KUKA KRL program: Kuka_Relative_Mo2.src

&ACCESS RVP
&REL 1
&PARAM TEMPLATE = C:\KRC\Roboter\Template\vorgabe
&PARAM EDITMASK = *
DEF Kuka_Relative_Mo2 ( )
; TOOL_DATA[1] = {FRAME: X 0.000,Y 0.000,Z 10.000,A 0.000,B 0.000,C 0.000}
$TOOL = {FRAME: X 0.000,Y 0.000,Z 10.000,A 0.000,B 0.000,C 0.000}
; $TOOL = TOOL_DATA[1]
; --------------------------
PTP {A1 -91.15290,A2 -57.66310,A3 113.87200,A4 27.68180,A5 -61.31820,A6 -12.21360}
; ---- Setting reference (Base) ----
$BASE = {FRAME: X 0.000,Y 0.000,Z 0.000,A 0.000,B 0.000,C 0.000}
; --------------------------
; ---- Setting tool (TCP) ----
; TOOL_DATA[1] = {FRAME: X 0.000,Y 0.000,Z 10.000,A 0.000,B 0.000,C 0.000}
$TOOL = {FRAME: X 0.000,Y 0.000,Z 10.000,A 0.000,B 0.000,C 0.000}
; $TOOL = TOOL_DATA[1]
; --------------------------
PTP {A1 -96.29580,A2 -57.85820,A3 114.83400,A4 -12.72140,A5 -60.67670,A6 8.34871}
; ---- Setting reference (Base) ----
$BASE = {FRAME: X 0.000,Y 0.000,Z 0.000,A 0.000,B 0.000,C 0.000}
; --------------------------
; ---- Setting tool (TCP) ----
; TOOL_DATA[1] = {FRAME: X 0.000,Y 0.000,Z 10.000,A 0.000,B 0.000,C 0.000}
$TOOL = {FRAME: X 0.000,Y 0.000,Z 10.000,A 0.000,B 0.000,C 0.000}
; $TOOL = TOOL_DATA[1]
; --------------------------
PTP {A1 -96.29580,A2 -57.85820,A3 114.83400,A4 -12.72140,A5 -60.67670,A6 -21.65130}
; ---- Setting reference (Base) ----
$BASE = {FRAME: X 0.000,Y 0.000,Z 0.000,A 0.000,B 0.000,C 0.000}
; --------------------------
; ---- Setting tool (TCP) ----
; TOOL_DATA[1] = {FRAME: X 0.000,Y 0.000,Z 10.000,A 0.000,B 0.000,C 0.000}
$TOOL = {FRAME: X 0.000,Y 0.000,Z 10.000,A 0.000,B 0.000,C 0.000}
; $TOOL = TOOL_DATA[1]
; --------------------------
PTP {A1 -96.29580,A2 -57.85820,A3 114.83400,A4 -12.72140,A5 -60.67670,A6 38.34870}
; ---- Setting reference (Base) ----
$BASE = {FRAME: X 0.000,Y 0.000,Z 0.000,A 0.000,B 0.000,C 0.000}
; --------------------------
; ---- Setting tool (TCP) ----
; TOOL_DATA[1] = {FRAME: X 0.000,Y 0.000,Z 10.000,A 0.000,B 0.000,C 0.000}
$TOOL = {FRAME: X 0.000,Y 0.000,Z 10.000,A 0.000,B 0.000,C 0.000}
; $TOOL = TOOL_DATA[1]
; --------------------------
PTP {A1 -96.29580,A2 -57.85820,A3 114.83400,A4 -12.72140,A5 -60.67670,A6 8.34871}
; ---- Setting reference (Base) ----
$BASE = {FRAME: X 0.000,Y 0.000,Z 0.000,A 0.000,B 0.000,C 0.000}
; --------------------------
; ---- Setting tool (TCP) ----
; TOOL_DATA[1] = {FRAME: X 0.000,Y 0.000,Z 10.000,A 0.000,B 0.000,C 0.000}
$TOOL = {FRAME: X 0.000,Y 0.000,Z 10.000,A 0.000,B 0.000,C 0.000}
; $TOOL = TOOL_DATA[1]
; --------------------------
PTP {A1 -85.43380,A2 -57.35410,A3 116.48600,A4 -0.25181,A5 -62.16390,A6 1.57543}
; ---- Setting reference (Base) ----
$BASE = {FRAME: X 0.000,Y 0.000,Z 0.000,A 0.000,B 0.000,C 0.000}
; --------------------------
; ---- Setting tool (TCP) ----
; TOOL_DATA[1] = {FRAME: X 0.000,Y 0.000,Z 10.000,A 0.000,B 0.000,C 0.000}
$TOOL = {FRAME: X 0.000,Y 0.000,Z 10.000,A 0.000,B 0.000,C 0.000}
; $TOOL = TOOL_DATA[1]
; --------------------------
PTP {A1 -90.40980,A2 -56.06330,A3 113.85800,A4 -38.62590,A5 -67.35010,A6 19.20140}
; ---- Setting reference (Base) ----
$BASE = {FRAME: X 0.000,Y 0.000,Z 0.000,A 0.000,B 0.000,C 0.000}
; --------------------------
; ---- Setting tool (TCP) ----
; TOOL_DATA[1] = {FRAME: X 0.000,Y 0.000,Z 10.000,A 0.000,B 0.000,C 0.000}
$TOOL = {FRAME: X 0.000,Y 0.000,Z 10.000,A 0.000,B 0.000,C 0.000}
; $TOOL = TOOL_DATA[1]
; --------------------------
PTP {A1 -80.44290,A2 -56.45170,A3 113.95500,A4 38.75120,A5 -65.60370,A6 -16.89390}
; ---- Setting reference (Base) ----
$BASE = {FRAME: X 0.000,Y 0.000,Z 0.000,A 0.000,B 0.000,C 0.000}
; --------------------------
; ---- Setting tool (TCP) ----
; TOOL_DATA[1] = {FRAME: X 0.000,Y 0.000,Z 10.000,A 0.000,B 0.000,C 0.000}
$TOOL = {FRAME: X 0.000,Y 0.000,Z 10.000,A 0.000,B 0.000,C 0.000}
; $TOOL = TOOL_DATA[1]
; --------------------------
PTP {A1 -85.43380,A2 -57.35410,A3 116.48600,A4 -0.25181,A5 -62.16390,A6 1.57543}
; ---- Setting reference (Base) ----
$BASE = {FRAME: X 0.000,Y 0.000,Z 0.000,A 0.000,B 0.000,C 0.000}
; --------------------------
; ---- Setting tool (TCP) ----
; TOOL_DATA[1] = {FRAME: X 0.000,Y 0.000,Z 10.000,A 0.000,B 0.000,C 0.000}
$TOOL = {FRAME: X 0.000,Y 0.000,Z 10.000,A 0.000,B 0.000,C 0.000}
; $TOOL = TOOL_DATA[1]
; --------------------------
PTP {A1 -85.43380,A2 -57.35410,A3 116.48600,A4 -0.25181,A5 -62.16390,A6 -28.42460}
; ---- Setting reference (Base) ----
$BASE = {FRAME: X 0.000,Y 0.000,Z 0.000,A 0.000,B 0.000,C 0.000}
; --------------------------
; ---- Setting tool (TCP) ----
; TOOL_DATA[1] = {FRAME: X 0.000,Y 0.000,Z 10.000,A 0.000,B 0.000,C 0.000}
$TOOL = {FRAME: X 0.000,Y 0.000,Z 10.000,A 0.000,B 0.000,C 0.000}
; $TOOL = TOOL_DATA[1]
; --------------------------
PTP {A1 -85.43380,A2 -57.35410,A3 116.48600,A4 -0.25181,A5 -62.16390,A6 31.57540}
; ---- Setting reference (Base) ----
$BASE = {FRAME: X 0.000,Y 0.000,Z 0.000,A 0.000,B 0.000,C 0.000}
; --------------------------
; ---- Setting tool (TCP) ----
; TOOL_DATA[1] = {FRAME: X 0.000,Y 0.000,Z 10.000,A 0.000,B 0.000,C 0.000}
$TOOL = {FRAME: X 0.000,Y 0.000,Z 10.000,A 0.000,B 0.000,C 0.000}
; $TOOL = TOOL_DATA[1]
; --------------------------
PTP {A1 -85.43380,A2 -57.35410,A3 116.48600,A4 -0.25181,A5 -62.16390,A6 1.57543}
; ---- Setting reference (Base) ----
$BASE = {FRAME: X 0.000,Y 0.000,Z 0.000,A 0.000,B 0.000,C 0.000}
; --------------------------
; ---- Setting tool (TCP) ----
; TOOL_DATA[1] = {FRAME: X 0.000,Y 0.000,Z 10.000,A 0.000,B 0.000,C 0.000}
$TOOL = {FRAME: X 0.000,Y 0.000,Z 10.000,A 0.000,B 0.000,C 0.000}
; $TOOL = TOOL_DATA[1]
; --------------------------
PTP {A1 -86.65140,A2 -57.29670,A3 116.45300,A4 -1.62638,A5 -62.19900,A6 2.28097}
; ---- Setting reference (Base) ----
$BASE = {FRAME: X 0.000,Y 0.000,Z 0.000,A 0.000,B 0.000,C 0.000}
; --------------------------
; ---- Setting tool (TCP) ----
; TOOL_DATA[1] = {FRAME: X 0.000,Y 0.000,Z 10.000,A 0.000,B 0.000,C 0.000}
$TOOL = {FRAME: X 0.000,Y 0.000,Z 10.000,A 0.000,B 0.000,C 0.000}
; $TOOL = TOOL_DATA[1]
; --------------------------
PTP {A1 -91.58690,A2 -55.92760,A3 113.65300,A4 -39.84090,A5 -67.69360,A6 19.77520}
; ---- Setting reference (Base) ----
$BASE = {FRAME: X 0.000,Y 0.000,Z 0.000,A 0.000,B 0.000,C 0.000}
; --------------------------
; ---- Setting tool (TCP) ----
; TOOL_DATA[1] = {FRAME: X 0.000,Y 0.000,Z 10.000,A 0.000,B 0.000,C 0.000}
$TOOL = {FRAME: X 0.000,Y 0.000,Z 10.000,A 0.000,B 0.000,C 0.000}
; $TOOL = TOOL_DATA[1]
; --------------------------
PTP {A1 -81.62640,A2 -56.47670,A3 114.09600,A4 37.49160,A5 -65.30300,A6 -16.26620}
; ---- Setting reference (Base) ----
$BASE = {FRAME: X 0.000,Y 0.000,Z 0.000,A 0.000,B 0.000,C 0.000}
; --------------------------
; ---- Setting tool (TCP) ----
; TOOL_DATA[1] = {FRAME: X 0.000,Y 0.000,Z 10.000,A 0.000,B 0.000,C 0.000}
$TOOL = {FRAME: X 0.000,Y 0.000,Z 10.000,A 0.000,B 0.000,C 0.000}
; $TOOL = TOOL_DATA[1]
; --------------------------
PTP {A1 -86.65140,A2 -57.29670,A3 116.45300,A4 -1.62638,A5 -62.19900,A6 2.28097}
; ---- Setting reference (Base) ----
$BASE = {FRAME: X 0.000,Y 0.000,Z 0.000,A 0.000,B 0.000,C 0.000}
; --------------------------
; ---- Setting tool (TCP) ----
; TOOL_DATA[1] = {FRAME: X 0.000,Y 0.000,Z 10.000,A 0.000,B 0.000,C 0.000}
$TOOL = {FRAME: X 0.000,Y 0.000,Z 10.000,A 0.000,B 0.000,C 0.000}
; $TOOL = TOOL_DATA[1]
; --------------------------
PTP {A1 -86.65140,A2 -57.29670,A3 116.45300,A4 -1.62638,A5 -62.19900,A6 -27.71900}
; ---- Setting reference (Base) ----
$BASE = {FRAME: X 0.000,Y 0.000,Z 0.000,A 0.000,B 0.000,C 0.000}
; --------------------------
; ---- Setting tool (TCP) ----
; TOOL_DATA[1] = {FRAME: X 0.000,Y 0.000,Z 10.000,A 0.000,B 0.000,C 0.000}
$TOOL = {FRAME: X 0.000,Y 0.000,Z 10.000,A 0.000,B 0.000,C 0.000}
; $TOOL = TOOL_DATA[1]
; --------------------------
PTP {A1 -86.65140,A2 -57.29670,A3 116.45300,A4 -1.62638,A5 -62.19900,A6 32.28100}
; ---- Setting reference (Base) ----
$BASE = {FRAME: X 0.000,Y 0.000,Z 0.000,A 0.000,B 0.000,C 0.000}
; --------------------------
; ---- Setting tool (TCP) ----
; TOOL_DATA[1] = {FRAME: X 0.000,Y 0.000,Z 10.000,A 0.000,B 0.000,C 0.000}
$TOOL = {FRAME: X 0.000,Y 0.000,Z 10.000,A 0.000,B 0.000,C 0.000}
; $TOOL = TOOL_DATA[1]
; --------------------------
PTP {A1 -86.65140,A2 -57.29670,A3 116.45300,A4 -1.62638,A5 -62.19900,A6 2.28097}
; ---- Setting reference (Base) ----
$BASE = {FRAME: X 0.000,Y 0.000,Z 0.000,A 0.000,B 0.000,C 0.000}
; --------------------------
; ---- Setting tool (TCP) ----
; TOOL_DATA[1] = {FRAME: X 0.000,Y 0.000,Z 10.000,A 0.000,B 0.000,C 0.000}
$TOOL = {FRAME: X 0.000,Y 0.000,Z 10.000,A 0.000,B 0.000,C 0.000}
; $TOOL = TOOL_DATA[1]
; --------------------------
PTP {A1 -87.86770,A2 -57.22000,A3 116.37900,A4 -2.99893,A5 -62.22640,A6 2.98512}
; ---- Setting reference (Base) ----
$BASE = {FRAME: X 0.000,Y 0.000,Z 0.000,A 0.000,B 0.000,C 0.000}
; --------------------------
; ---- Setting tool (TCP) ----
; TOOL_DATA[1] = {FRAME: X 0.000,Y 0.000,Z 10.000,A 0.000,B 0.000,C 0.000}
$TOOL = {FRAME: X 0.000,Y 0.000,Z 10.000,A 0.000,B 0.000,C 0.000}
; $TOOL = TOOL_DATA[1]
; --------------------------
PTP {A1 -92.75860,A2 -55.77320,A3 113.40700,A4 -41.04920,A5 -68.03040,A6 20.35390}
; ---- Setting reference (Base) ----
$BASE = {FRAME: X 0.000,Y 0.000,Z 0.000,A 0.000,B 0.000,C 0.000}
; --------------------------
; ---- Setting tool (TCP) ----
; TOOL_DATA[1] = {FRAME: X 0.000,Y 0.000,Z 10.000,A 0.000,B 0.000,C 0.000}
$TOOL = {FRAME: X 0.000,Y 0.000,Z 10.000,A 0.000,B 0.000,C 0.000}
; $TOOL = TOOL_DATA[1]
; --------------------------
PTP {A1 -82.81280,A2 -56.48220,A3 114.19600,A4 36.22780,A5 -64.99770,A6 -15.64440}
; ---- Setting reference (Base) ----
$BASE = {FRAME: X 0.000,Y 0.000,Z 0.000,A 0.000,B 0.000,C 0.000}
; --------------------------
; ---- Setting tool (TCP) ----
; TOOL_DATA[1] = {FRAME: X 0.000,Y 0.000,Z 10.000,A 0.000,B 0.000,C 0.000}
$TOOL = {FRAME: X 0.000,Y 0.000,Z 10.000,A 0.000,B 0.000,C 0.000}
; $TOOL = TOOL_DATA[1]
; --------------------------
PTP {A1 -87.86770,A2 -57.22000,A3 116.37900,A4 -2.99893,A5 -62.22640,A6 2.98512}
; ---- Setting reference (Base) ----
$BASE = {FRAME: X 0.000,Y 0.000,Z 0.000,A 0.000,B 0.000,C 0.000}
; --------------------------
; ---- Setting tool (TCP) ----
; TOOL_DATA[1] = {FRAME: X 0.000,Y 0.000,Z 10.000,A 0.000,B 0.000,C 0.000}
$TOOL = {FRAME: X 0.000,Y 0.000,Z 10.000,A 0.000,B 0.000,C 0.000}
; $TOOL = TOOL_DATA[1]
; --------------------------
PTP {A1 -87.86770,A2 -57.22000,A3 116.37900,A4 -2.99893,A5 -62.22640,A6 -27.01490}
; ---- Setting reference (Base) ----
$BASE = {FRAME: X 0.000,Y 0.000,Z 0.000,A 0.000,B 0.000,C 0.000}
; --------------------------
; ---- Setting tool (TCP) ----
; TOOL_DATA[1] = {FRAME: X 0.000,Y 0.000,Z 10.000,A 0.000,B 0.000,C 0.000}
$TOOL = {FRAME: X 0.000,Y 0.000,Z 10.000,A 0.000,B 0.000,C 0.000}
; $TOOL = TOOL_DATA[1]
; --------------------------
PTP {A1 -87.86770,A2 -57.22000,A3 116.37900,A4 -2.99893,A5 -62.22640,A6 32.98510}
; ---- Setting reference (Base) ----
$BASE = {FRAME: X 0.000,Y 0.000,Z 0.000,A 0.000,B 0.000,C 0.000}
; --------------------------
; ---- Setting tool (TCP) ----
; TOOL_DATA[1] = {FRAME: X 0.000,Y 0.000,Z 10.000,A 0.000,B 0.000,C 0.000}
$TOOL = {FRAME: X 0.000,Y 0.000,Z 10.000,A 0.000,B 0.000,C 0.000}
; $TOOL = TOOL_DATA[1]
; --------------------------
PTP {A1 -87.86770,A2 -57.22000,A3 116.37900,A4 -2.99893,A5 -62.22640,A6 2.98512}
; ---- Setting reference (Base) ----
$BASE = {FRAME: X 0.000,Y 0.000,Z 0.000,A 0.000,B 0.000,C 0.000}
; --------------------------
; ---- Setting tool (TCP) ----
; TOOL_DATA[1] = {FRAME: X 0.000,Y 0.000,Z 10.000,A 0.000,B 0.000,C 0.000}
$TOOL = {FRAME: X 0.000,Y 0.000,Z 10.000,A 0.000,B 0.000,C 0.000}
; $TOOL = TOOL_DATA[1]
; --------------------------
PTP {A1 -89.08150,A2 -57.12440,A3 116.26300,A4 -4.36870,A5 -62.24600,A6 3.68858}
; ---- Setting reference (Base) ----
$BASE = {FRAME: X 0.000,Y 0.000,Z 0.000,A 0.000,B 0.000,C 0.000}
; --------------------------
; ---- Setting tool (TCP) ----
; TOOL_DATA[1] = {FRAME: X 0.000,Y 0.000,Z 10.000,A 0.000,B 0.000,C 0.000}
$TOOL = {FRAME: X 0.000,Y 0.000,Z 10.000,A 0.000,B 0.000,C 0.000}
; $TOOL = TOOL_DATA[1]
; --------------------------
PTP {A1 -93.92390,A2 -55.60020,A3 113.12000,A4 -42.24980,A5 -68.36080,A6 20.93800}
; ---- Setting reference (Base) ----
$BASE = {FRAME: X 0.000,Y 0.000,Z 0.000,A 0.000,B 0.000,C 0.000}
; --------------------------
; ---- Setting tool (TCP) ----
; TOOL_DATA[1] = {FRAME: X 0.000,Y 0.000,Z 10.000,A 0.000,B 0.000,C 0.000}
$TOOL = {FRAME: X 0.000,Y 0.000,Z 10.000,A 0.000,B 0.000,C 0.000}
; $TOOL = TOOL_DATA[1]
; --------------------------
PTP {A1 -84.00130,A2 -56.46850,A3 114.25400,A4 34.96070,A5 -64.68740,A6 -15.02820}
; ---- Setting reference (Base) ----
$BASE = {FRAME: X 0.000,Y 0.000,Z 0.000,A 0.000,B 0.000,C 0.000}
; --------------------------
; ---- Setting tool (TCP) ----
; TOOL_DATA[1] = {FRAME: X 0.000,Y 0.000,Z 10.000,A 0.000,B 0.000,C 0.000}
$TOOL = {FRAME: X 0.000,Y 0.000,Z 10.000,A 0.000,B 0.000,C 0.000}
; $TOOL = TOOL_DATA[1]
; --------------------------
PTP {A1 -89.08150,A2 -57.12440,A3 116.26300,A4 -4.36870,A5 -62.24600,A6 3.68858}
; ---- Setting reference (Base) ----
$BASE = {FRAME: X 0.000,Y 0.000,Z 0.000,A 0.000,B 0.000,C 0.000}
; --------------------------
; ---- Setting tool (TCP) ----
; TOOL_DATA[1] = {FRAME: X 0.000,Y 0.000,Z 10.000,A 0.000,B 0.000,C 0.000}
$TOOL = {FRAME: X 0.000,Y 0.000,Z 10.000,A 0.000,B 0.000,C 0.000}
; $TOOL = TOOL_DATA[1]
; --------------------------
PTP {A1 -89.08150,A2 -57.12440,A3 116.26300,A4 -4.36870,A5 -62.24600,A6 -26.31140}
; ---- Setting reference (Base) ----
$BASE = {FRAME: X 0.000,Y 0.000,Z 0.000,A 0.000,B 0.000,C 0.000}
; --------------------------
; ---- Setting tool (TCP) ----
; TOOL_DATA[1] = {FRAME: X 0.000,Y 0.000,Z 10.000,A 0.000,B 0.000,C 0.000}
$TOOL = {FRAME: X 0.000,Y 0.000,Z 10.000,A 0.000,B 0.000,C 0.000}
; $TOOL = TOOL_DATA[1]
; --------------------------
PTP {A1 -89.08150,A2 -57.12440,A3 116.26300,A4 -4.36870,A5 -62.24600,A6 33.68860}
; ---- Setting reference (Base) ----
$BASE = {FRAME: X 0.000,Y 0.000,Z 0.000,A 0.000,B 0.000,C 0.000}
; --------------------------
; ---- Setting tool (TCP) ----
; TOOL_DATA[1] = {FRAME: X 0.000,Y 0.000,Z 10.000,A 0.000,B 0.000,C 0.000}
$TOOL = {FRAME: X 0.000,Y 0.000,Z 10.000,A 0.000,B 0.000,C 0.000}
; $TOOL = TOOL_DATA[1]
; --------------------------
PTP {A1 -89.08150,A2 -57.12440,A3 116.26300,A4 -4.36870,A5 -62.24600,A6 3.68858}
; ---- Setting reference (Base) ----
$BASE = {FRAME: X 0.000,Y 0.000,Z 0.000,A 0.000,B 0.000,C 0.000}
; --------------------------
; ---- Setting tool (TCP) ----
; TOOL_DATA[1] = {FRAME: X 0.000,Y 0.000,Z 10.000,A 0.000,B 0.000,C 0.000}
$TOOL = {FRAME: X 0.000,Y 0.000,Z 10.000,A 0.000,B 0.000,C 0.000}
; $TOOL = TOOL_DATA[1]
; --------------------------
PTP {A1 -90.29180,A2 -57.00970,A3 116.10500,A4 -5.73493,A5 -62.25790,A6 4.39206}
; ---- Setting reference (Base) ----
$BASE = {FRAME: X 0.000,Y 0.000,Z 0.000,A 0.000,B 0.000,C 0.000}
; --------------------------
; ---- Setting tool (TCP) ----
; TOOL_DATA[1] = {FRAME: X 0.000,Y 0.000,Z 10.000,A 0.000,B 0.000,C 0.000}
$TOOL = {FRAME: X 0.000,Y 0.000,Z 10.000,A 0.000,B 0.000,C 0.000}
; $TOOL = TOOL_DATA[1]
; --------------------------
PTP {A1 -95.08190,A2 -55.40870,A3 112.79300,A4 -43.44190,A5 -68.68500,A6 21.52800}
; ---- Setting reference (Base) ----
$BASE = {FRAME: X 0.000,Y 0.000,Z 0.000,A 0.000,B 0.000,C 0.000}
; --------------------------
; ---- Setting tool (TCP) ----
; TOOL_DATA[1] = {FRAME: X 0.000,Y 0.000,Z 10.000,A 0.000,B 0.000,C 0.000}
$TOOL = {FRAME: X 0.000,Y 0.000,Z 10.000,A 0.000,B 0.000,C 0.000}
; $TOOL = TOOL_DATA[1]
; --------------------------
PTP {A1 -85.19070,A2 -56.43550,A3 114.27100,A4 33.69130,A5 -64.37170,A6 -14.41710}
; ---- Setting reference (Base) ----
$BASE = {FRAME: X 0.000,Y 0.000,Z 0.000,A 0.000,B 0.000,C 0.000}
; --------------------------
; ---- Setting tool (TCP) ----
; TOOL_DATA[1] = {FRAME: X 0.000,Y 0.000,Z 10.000,A 0.000,B 0.000,C 0.000}
$TOOL = {FRAME: X 0.000,Y 0.000,Z 10.000,A 0.000,B 0.000,C 0.000}
; $TOOL = TOOL_DATA[1]
; --------------------------
PTP {A1 -90.29180,A2 -57.00970,A3 116.10500,A4 -5.73493,A5 -62.25790,A6 4.39206}
; ---- Setting reference (Base) ----
$BASE = {FRAME: X 0.000,Y 0.000,Z 0.000,A 0.000,B 0.000,C 0.000}
; --------------------------
; ---- Setting tool (TCP) ----
; TOOL_DATA[1] = {FRAME: X 0.000,Y 0.000,Z 10.000,A 0.000,B 0.000,C 0.000}
$TOOL = {FRAME: X 0.000,Y 0.000,Z 10.000,A 0.000,B 0.000,C 0.000}
; $TOOL = TOOL_DATA[1]
; --------------------------
PTP {A1 -90.29180,A2 -57.00970,A3 116.10500,A4 -5.73493,A5 -62.25790,A6 -25.60790}
; ---- Setting reference (Base) ----
$BASE = {FRAME: X 0.000,Y 0.000,Z 0.000,A 0.000,B 0.000,C 0.000}
; --------------------------
; ---- Setting tool (TCP) ----
; TOOL_DATA[1] = {FRAME: X 0.000,Y 0.000,Z 10.000,A 0.000,B 0.000,C 0.000}
$TOOL = {FRAME: X 0.000,Y 0.000,Z 10.000,A 0.000,B 0.000,C 0.000}
; $TOOL = TOOL_DATA[1]
; --------------------------
PTP {A1 -90.29180,A2 -57.00970,A3 116.10500,A4 -5.73493,A5 -62.25790,A6 34.39210}
; ---- Setting reference (Base) ----
$BASE = {FRAME: X 0.000,Y 0.000,Z 0.000,A 0.000,B 0.000,C 0.000}
; --------------------------
; ---- Setting tool (TCP) ----
; TOOL_DATA[1] = {FRAME: X 0.000,Y 0.000,Z 10.000,A 0.000,B 0.000,C 0.000}
$TOOL = {FRAME: X 0.000,Y 0.000,Z 10.000,A 0.000,B 0.000,C 0.000}
; $TOOL = TOOL_DATA[1]
; --------------------------
PTP {A1 -90.29180,A2 -57.00970,A3 116.10500,A4 -5.73493,A5 -62.25790,A6 4.39206}
; ---- Setting reference (Base) ----
$BASE = {FRAME: X 0.000,Y 0.000,Z 0.000,A 0.000,B 0.000,C 0.000}
; --------------------------
; ---- Setting tool (TCP) ----
; TOOL_DATA[1] = {FRAME: X 0.000,Y 0.000,Z 10.000,A 0.000,B 0.000,C 0.000}
$TOOL = {FRAME: X 0.000,Y 0.000,Z 10.000,A 0.000,B 0.000,C 0.000}
; $TOOL = TOOL_DATA[1]
; --------------------------
PTP {A1 -91.49750,A2 -56.87630,A3 115.90600,A4 -7.09688,A5 -62.26190,A6 5.09629}
; ---- Setting reference (Base) ----
$BASE = {FRAME: X 0.000,Y 0.000,Z 0.000,A 0.000,B 0.000,C 0.000}
; --------------------------
; ---- Setting tool (TCP) ----
; TOOL_DATA[1] = {FRAME: X 0.000,Y 0.000,Z 10.000,A 0.000,B 0.000,C 0.000}
$TOOL = {FRAME: X 0.000,Y 0.000,Z 10.000,A 0.000,B 0.000,C 0.000}
; $TOOL = TOOL_DATA[1]
; --------------------------
PTP {A1 -96.23170,A2 -55.19870,A3 112.42600,A4 -44.62480,A5 -69.00340,A6 22.12420}
; ---- Setting reference (Base) ----
$BASE = {FRAME: X 0.000,Y 0.000,Z 0.000,A 0.000,B 0.000,C 0.000}
; --------------------------
; ---- Setting tool (TCP) ----
; TOOL_DATA[1] = {FRAME: X 0.000,Y 0.000,Z 10.000,A 0.000,B 0.000,C 0.000}
$TOOL = {FRAME: X 0.000,Y 0.000,Z 10.000,A 0.000,B 0.000,C 0.000}
; $TOOL = TOOL_DATA[1]
; --------------------------
PTP {A1 -86.38010,A2 -56.38330,A3 114.24800,A4 32.42060,A5 -64.05010,A6 -13.81090}
; ---- Setting reference (Base) ----
$BASE = {FRAME: X 0.000,Y 0.000,Z 0.000,A 0.000,B 0.000,C 0.000}
; --------------------------
; ---- Setting tool (TCP) ----
; TOOL_DATA[1] = {FRAME: X 0.000,Y 0.000,Z 10.000,A 0.000,B 0.000,C 0.000}
$TOOL = {FRAME: X 0.000,Y 0.000,Z 10.000,A 0.000,B 0.000,C 0.000}
; $TOOL = TOOL_DATA[1]
; --------------------------
PTP {A1 -91.49750,A2 -56.87630,A3 115.90600,A4 -7.09688,A5 -62.26190,A6 5.09629}
; ---- Setting reference (Base) ----
$BASE = {FRAME: X 0.000,Y 0.000,Z 0.000,A 0.000,B 0.000,C 0.000}
; --------------------------
; ---- Setting tool (TCP) ----
; TOOL_DATA[1] = {FRAME: X 0.000,Y 0.000,Z 10.000,A 0.000,B 0.000,C 0.000}
$TOOL = {FRAME: X 0.000,Y 0.000,Z 10.000,A 0.000,B 0.000,C 0.000}
; $TOOL = TOOL_DATA[1]
; --------------------------
PTP {A1 -91.49750,A2 -56.87630,A3 115.90600,A4 -7.09688,A5 -62.26190,A6 -24.90370}
; ---- Setting reference (Base) ----
$BASE = {FRAME: X 0.000,Y 0.000,Z 0.000,A 0.000,B 0.000,C 0.000}
; --------------------------
; ---- Setting tool (TCP) ----
; TOOL_DATA[1] = {FRAME: X 0.000,Y 0.000,Z 10.000,A 0.000,B 0.000,C 0.000}
$TOOL = {FRAME: X 0.000,Y 0.000,Z 10.000,A 0.000,B 0.000,C 0.000}
; $TOOL = TOOL_DATA[1]
; --------------------------
PTP {A1 -91.49750,A2 -56.87630,A3 115.90600,A4 -7.09688,A5 -62.26190,A6 35.09630}
; ---- Setting reference (Base) ----
$BASE = {FRAME: X 0.000,Y 0.000,Z 0.000,A 0.000,B 0.000,C 0.000}
; --------------------------
; ---- Setting tool (TCP) ----
; TOOL_DATA[1] = {FRAME: X 0.000,Y 0.000,Z 10.000,A 0.000,B 0.000,C 0.000}
$TOOL = {FRAME: X 0.000,Y 0.000,Z 10.000,A 0.000,B 0.000,C 0.000}
; $TOOL = TOOL_DATA[1]
; --------------------------
PTP {A1 -91.49750,A2 -56.87630,A3 115.90600,A4 -7.09688,A5 -62.26190,A6 5.09629}
; ---- Setting reference (Base) ----
$BASE = {FRAME: X 0.000,Y 0.000,Z 0.000,A 0.000,B 0.000,C 0.000}
; --------------------------
; ---- Setting tool (TCP) ----
; TOOL_DATA[1] = {FRAME: X 0.000,Y 0.000,Z 10.000,A 0.000,B 0.000,C 0.000}
$TOOL = {FRAME: X 0.000,Y 0.000,Z 10.000,A 0.000,B 0.000,C 0.000}
; $TOOL = TOOL_DATA[1]
; --------------------------
PTP {A1 -92.69750,A2 -56.72400,A3 115.66600,A4 -8.45384,A5 -62.25820,A6 5.80196}
; ---- Setting reference (Base) ----
$BASE = {FRAME: X 0.000,Y 0.000,Z 0.000,A 0.000,B 0.000,C 0.000}
; --------------------------
; ---- Setting tool (TCP) ----
; TOOL_DATA[1] = {FRAME: X 0.000,Y 0.000,Z 10.000,A 0.000,B 0.000,C 0.000}
$TOOL = {FRAME: X 0.000,Y 0.000,Z 10.000,A 0.000,B 0.000,C 0.000}
; $TOOL = TOOL_DATA[1]
; --------------------------
PTP {A1 -97.37260,A2 -54.97050,A3 112.01800,A4 -45.79760,A5 -69.31630,A6 22.72710}
; ---- Setting reference (Base) ----
$BASE = {FRAME: X 0.000,Y 0.000,Z 0.000,A 0.000,B 0.000,C 0.000}
; --------------------------
; ---- Setting tool (TCP) ----
; TOOL_DATA[1] = {FRAME: X 0.000,Y 0.000,Z 10.000,A 0.000,B 0.000,C 0.000}
$TOOL = {FRAME: X 0.000,Y 0.000,Z 10.000,A 0.000,B 0.000,C 0.000}
; $TOOL = TOOL_DATA[1]
; --------------------------
PTP {A1 -87.56840,A2 -56.31190,A3 114.18200,A4 31.14940,A5 -63.72240,A6 -13.20900}
; ---- Setting reference (Base) ----
$BASE = {FRAME: X 0.000,Y 0.000,Z 0.000,A 0.000,B 0.000,C 0.000}
; --------------------------
; ---- Setting tool (TCP) ----
; TOOL_DATA[1] = {FRAME: X 0.000,Y 0.000,Z 10.000,A 0.000,B 0.000,C 0.000}
$TOOL = {FRAME: X 0.000,Y 0.000,Z 10.000,A 0.000,B 0.000,C 0.000}
; $TOOL = TOOL_DATA[1]
; --------------------------
PTP {A1 -92.69750,A2 -56.72400,A3 115.66600,A4 -8.45384,A5 -62.25820,A6 5.80196}
; ---- Setting reference (Base) ----
$BASE = {FRAME: X 0.000,Y 0.000,Z 0.000,A 0.000,B 0.000,C 0.000}
; --------------------------
; ---- Setting tool (TCP) ----
; TOOL_DATA[1] = {FRAME: X 0.000,Y 0.000,Z 10.000,A 0.000,B 0.000,C 0.000}
$TOOL = {FRAME: X 0.000,Y 0.000,Z 10.000,A 0.000,B 0.000,C 0.000}
; $TOOL = TOOL_DATA[1]
; --------------------------
PTP {A1 -92.69750,A2 -56.72400,A3 115.66600,A4 -8.45384,A5 -62.25820,A6 -24.19800}
; ---- Setting reference (Base) ----
$BASE = {FRAME: X 0.000,Y 0.000,Z 0.000,A 0.000,B 0.000,C 0.000}
; --------------------------
; ---- Setting tool (TCP) ----
; TOOL_DATA[1] = {FRAME: X 0.000,Y 0.000,Z 10.000,A 0.000,B 0.000,C 0.000}
$TOOL = {FRAME: X 0.000,Y 0.000,Z 10.000,A 0.000,B 0.000,C 0.000}
; $TOOL = TOOL_DATA[1]
; --------------------------
PTP {A1 -92.69750,A2 -56.72400,A3 115.66600,A4 -8.45384,A5 -62.25820,A6 35.80200}
; ---- Setting reference (Base) ----
$BASE = {FRAME: X 0.000,Y 0.000,Z 0.000,A 0.000,B 0.000,C 0.000}
; --------------------------
; ---- Setting tool (TCP) ----
; TOOL_DATA[1] = {FRAME: X 0.000,Y 0.000,Z 10.000,A 0.000,B 0.000,C 0.000}
$TOOL = {FRAME: X 0.000,Y 0.000,Z 10.000,A 0.000,B 0.000,C 0.000}
; $TOOL = TOOL_DATA[1]
; --------------------------
PTP {A1 -92.69750,A2 -56.72400,A3 115.66600,A4 -8.45384,A5 -62.25820,A6 5.80196}
; ---- Setting reference (Base) ----
$BASE = {FRAME: X 0.000,Y 0.000,Z 0.000,A 0.000,B 0.000,C 0.000}
; --------------------------
; ---- Setting tool (TCP) ----
; TOOL_DATA[1] = {FRAME: X 0.000,Y 0.000,Z 10.000,A 0.000,B 0.000,C 0.000}
$TOOL = {FRAME: X 0.000,Y 0.000,Z 10.000,A 0.000,B 0.000,C 0.000}
; $TOOL = TOOL_DATA[1]
; --------------------------
PTP {A1 -93.89100,A2 -56.55310,A3 115.38400,A4 -9.80514,A5 -62.24670,A6 6.50979}
; ---- Setting reference (Base) ----
$BASE = {FRAME: X 0.000,Y 0.000,Z 0.000,A 0.000,B 0.000,C 0.000}
; --------------------------
; ---- Setting tool (TCP) ----
; TOOL_DATA[1] = {FRAME: X 0.000,Y 0.000,Z 10.000,A 0.000,B 0.000,C 0.000}
$TOOL = {FRAME: X 0.000,Y 0.000,Z 10.000,A 0.000,B 0.000,C 0.000}
; $TOOL = TOOL_DATA[1]
; --------------------------
PTP {A1 -98.50370,A2 -54.72400,A3 111.57000,A4 -46.95960,A5 -69.62410,A6 23.33710}
; ---- Setting reference (Base) ----
$BASE = {FRAME: X 0.000,Y 0.000,Z 0.000,A 0.000,B 0.000,C 0.000}
; --------------------------
; ---- Setting tool (TCP) ----
; TOOL_DATA[1] = {FRAME: X 0.000,Y 0.000,Z 10.000,A 0.000,B 0.000,C 0.000}
$TOOL = {FRAME: X 0.000,Y 0.000,Z 10.000,A 0.000,B 0.000,C 0.000}
; $TOOL = TOOL_DATA[1]
; --------------------------
PTP {A1 -88.75460,A2 -56.22160,A3 114.07600,A4 29.87860,A5 -63.38820,A6 -12.61090}
; ---- Setting reference (Base) ----
$BASE = {FRAME: X 0.000,Y 0.000,Z 0.000,A 0.000,B 0.000,C 0.000}
; --------------------------
; ---- Setting tool (TCP) ----
; TOOL_DATA[1] = {FRAME: X 0.000,Y 0.000,Z 10.000,A 0.000,B 0.000,C 0.000}
$TOOL = {FRAME: X 0.000,Y 0.000,Z 10.000,A 0.000,B 0.000,C 0.000}
; $TOOL = TOOL_DATA[1]
; --------------------------
PTP {A1 -93.89100,A2 -56.55310,A3 115.38400,A4 -9.80514,A5 -62.24670,A6 6.50979}
; ---- Setting reference (Base) ----
$BASE = {FRAME: X 0.000,Y 0.000,Z 0.000,A 0.000,B 0.000,C 0.000}
; --------------------------
; ---- Setting tool (TCP) ----
; TOOL_DATA[1] = {FRAME: X 0.000,Y 0.000,Z 10.000,A 0.000,B 0.000,C 0.000}
$TOOL = {FRAME: X 0.000,Y 0.000,Z 10.000,A 0.000,B 0.000,C 0.000}
; $TOOL = TOOL_DATA[1]
; --------------------------
PTP {A1 -93.89100,A2 -56.55310,A3 115.38400,A4 -9.80514,A5 -62.24670,A6 -23.49020}
; ---- Setting reference (Base) ----
$BASE = {FRAME: X 0.000,Y 0.000,Z 0.000,A 0.000,B 0.000,C 0.000}
; --------------------------
; ---- Setting tool (TCP) ----
; TOOL_DATA[1] = {FRAME: X 0.000,Y 0.000,Z 10.000,A 0.000,B 0.000,C 0.000}
$TOOL = {FRAME: X 0.000,Y 0.000,Z 10.000,A 0.000,B 0.000,C 0.000}
; $TOOL = TOOL_DATA[1]
; --------------------------
PTP {A1 -93.89100,A2 -56.55310,A3 115.38400,A4 -9.80514,A5 -62.24670,A6 36.50980}
; ---- Setting reference (Base) ----
$BASE = {FRAME: X 0.000,Y 0.000,Z 0.000,A 0.000,B 0.000,C 0.000}
; --------------------------
; ---- Setting tool (TCP) ----
; TOOL_DATA[1] = {FRAME: X 0.000,Y 0.000,Z 10.000,A 0.000,B 0.000,C 0.000}
$TOOL = {FRAME: X 0.000,Y 0.000,Z 10.000,A 0.000,B 0.000,C 0.000}
; $TOOL = TOOL_DATA[1]
; --------------------------
PTP {A1 -93.89100,A2 -56.55310,A3 115.38400,A4 -9.80514,A5 -62.24670,A6 6.50979}
; ---- Setting reference (Base) ----
$BASE = {FRAME: X 0.000,Y 0.000,Z 0.000,A 0.000,B 0.000,C 0.000}
; --------------------------
; ---- Setting tool (TCP) ----
; TOOL_DATA[1] = {FRAME: X 0.000,Y 0.000,Z 10.000,A 0.000,B 0.000,C 0.000}
$TOOL = {FRAME: X 0.000,Y 0.000,Z 10.000,A 0.000,B 0.000,C 0.000}
; $TOOL = TOOL_DATA[1]
; --------------------------
PTP {A1 -95.07680,A2 -56.36370,A3 115.06100,A4 -11.15010,A5 -62.22750,A6 7.22049}
; ---- Setting reference (Base) ----
$BASE = {FRAME: X 0.000,Y 0.000,Z 0.000,A 0.000,B 0.000,C 0.000}
; --------------------------
; ---- Setting tool (TCP) ----
; TOOL_DATA[1] = {FRAME: X 0.000,Y 0.000,Z 10.000,A 0.000,B 0.000,C 0.000}
$TOOL = {FRAME: X 0.000,Y 0.000,Z 10.000,A 0.000,B 0.000,C 0.000}
; $TOOL = TOOL_DATA[1]
; --------------------------
PTP {A1 -99.62430,A2 -54.45930,A3 111.08300,A4 -48.11000,A5 -69.92710,A6 23.95460}
; ---- Setting reference (Base) ----
$BASE = {FRAME: X 0.000,Y 0.000,Z 0.000,A 0.000,B 0.000,C 0.000}
; --------------------------
; ---- Setting tool (TCP) ----
; TOOL_DATA[1] = {FRAME: X 0.000,Y 0.000,Z 10.000,A 0.000,B 0.000,C 0.000}
$TOOL = {FRAME: X 0.000,Y 0.000,Z 10.000,A 0.000,B 0.000,C 0.000}
; $TOOL = TOOL_DATA[1]
; --------------------------
PTP {A1 -89.93770,A2 -56.11230,A3 113.92800,A4 28.60910,A5 -63.04720,A6 -12.01630}
; ---- Setting reference (Base) ----
$BASE = {FRAME: X 0.000,Y 0.000,Z 0.000,A 0.000,B 0.000,C 0.000}
; --------------------------
; ---- Setting tool (TCP) ----
; TOOL_DATA[1] = {FRAME: X 0.000,Y 0.000,Z 10.000,A 0.000,B 0.000,C 0.000}
$TOOL = {FRAME: X 0.000,Y 0.000,Z 10.000,A 0.000,B 0.000,C 0.000}
; $TOOL = TOOL_DATA[1]
; --------------------------
PTP {A1 -95.07680,A2 -56.36370,A3 115.06100,A4 -11.15010,A5 -62.22750,A6 7.22049}
; ---- Setting reference (Base) ----
$BASE = {FRAME: X 0.000,Y 0.000,Z 0.000,A 0.000,B 0.000,C 0.000}
; --------------------------
; ---- Setting tool (TCP) ----
; TOOL_DATA[1] = {FRAME: X 0.000,Y 0.000,Z 10.000,A 0.000,B 0.000,C 0.000}
$TOOL = {FRAME: X 0.000,Y 0.000,Z 10.000,A 0.000,B 0.000,C 0.000}
; $TOOL = TOOL_DATA[1]
; --------------------------
PTP {A1 -95.07680,A2 -56.36370,A3 115.06100,A4 -11.15010,A5 -62.22750,A6 -22.77950}
; ---- Setting reference (Base) ----
$BASE = {FRAME: X 0.000,Y 0.000,Z 0.000,A 0.000,B 0.000,C 0.000}
; --------------------------
; ---- Setting tool (TCP) ----
; TOOL_DATA[1] = {FRAME: X 0.000,Y 0.000,Z 10.000,A 0.000,B 0.000,C 0.000}
$TOOL = {FRAME: X 0.000,Y 0.000,Z 10.000,A 0.000,B 0.000,C 0.000}
; $TOOL = TOOL_DATA[1]
; --------------------------
PTP {A1 -95.07680,A2 -56.36370,A3 115.06100,A4 -11.15010,A5 -62.22750,A6 37.22050}
; ---- Setting reference (Base) ----
$BASE = {FRAME: X 0.000,Y 0.000,Z 0.000,A 0.000,B 0.000,C 0.000}
; --------------------------
; ---- Setting tool (TCP) ----
; TOOL_DATA[1] = {FRAME: X 0.000,Y 0.000,Z 10.000,A 0.000,B 0.000,C 0.000}
$TOOL = {FRAME: X 0.000,Y 0.000,Z 10.000,A 0.000,B 0.000,C 0.000}
; $TOOL = TOOL_DATA[1]
; --------------------------
PTP {A1 -95.07680,A2 -56.36370,A3 115.06100,A4 -11.15010,A5 -62.22750,A6 7.22049}
; ---- Setting reference (Base) ----
$BASE = {FRAME: X 0.000,Y 0.000,Z 0.000,A 0.000,B 0.000,C 0.000}
; --------------------------
; ---- Setting tool (TCP) ----
; TOOL_DATA[1] = {FRAME: X 0.000,Y 0.000,Z 10.000,A 0.000,B 0.000,C 0.000}
$TOOL = {FRAME: X 0.000,Y 0.000,Z 10.000,A 0.000,B 0.000,C 0.000}
; $TOOL = TOOL_DATA[1]
; --------------------------
PTP {A1 -96.25400,A2 -56.15580,A3 114.69800,A4 -12.48820,A5 -62.20070,A6 7.93472}
; ---- Setting reference (Base) ----
$BASE = {FRAME: X 0.000,Y 0.000,Z 0.000,A 0.000,B 0.000,C 0.000}
; --------------------------
; ---- Setting tool (TCP) ----
; TOOL_DATA[1] = {FRAME: X 0.000,Y 0.000,Z 10.000,A 0.000,B 0.000,C 0.000}
$TOOL = {FRAME: X 0.000,Y 0.000,Z 10.000,A 0.000,B 0.000,C 0.000}
; $TOOL = TOOL_DATA[1]
; --------------------------
PTP {A1 -100.73400,A2 -54.17670,A3 110.55600,A4 -49.24820,A5 -70.22560,A6 24.57980}
; ---- Setting reference (Base) ----
$BASE = {FRAME: X 0.000,Y 0.000,Z 0.000,A 0.000,B 0.000,C 0.000}
; --------------------------
; ---- Setting tool (TCP) ----
; TOOL_DATA[1] = {FRAME: X 0.000,Y 0.000,Z 10.000,A 0.000,B 0.000,C 0.000}
$TOOL = {FRAME: X 0.000,Y 0.000,Z 10.000,A 0.000,B 0.000,C 0.000}
; $TOOL = TOOL_DATA[1]
; --------------------------
PTP {A1 -91.11670,A2 -55.98410,A3 113.74000,A4 27.34170,A5 -62.69900,A6 -11.42440}
; ---- Setting reference (Base) ----
$BASE = {FRAME: X 0.000,Y 0.000,Z 0.000,A 0.000,B 0.000,C 0.000}
; --------------------------
; ---- Setting tool (TCP) ----
; TOOL_DATA[1] = {FRAME: X 0.000,Y 0.000,Z 10.000,A 0.000,B 0.000,C 0.000}
$TOOL = {FRAME: X 0.000,Y 0.000,Z 10.000,A 0.000,B 0.000,C 0.000}
; $TOOL = TOOL_DATA[1]
; --------------------------
PTP {A1 -96.25400,A2 -56.15580,A3 114.69800,A4 -12.48820,A5 -62.20070,A6 7.93472}
; ---- Setting reference (Base) ----
$BASE = {FRAME: X 0.000,Y 0.000,Z 0.000,A 0.000,B 0.000,C 0.000}
; --------------------------
; ---- Setting tool (TCP) ----
; TOOL_DATA[1] = {FRAME: X 0.000,Y 0.000,Z 10.000,A 0.000,B 0.000,C 0.000}
$TOOL = {FRAME: X 0.000,Y 0.000,Z 10.000,A 0.000,B 0.000,C 0.000}
; $TOOL = TOOL_DATA[1]
; --------------------------
PTP {A1 -96.25400,A2 -56.15580,A3 114.69800,A4 -12.48820,A5 -62.20070,A6 -22.06530}
; ---- Setting reference (Base) ----
$BASE = {FRAME: X 0.000,Y 0.000,Z 0.000,A 0.000,B 0.000,C 0.000}
; --------------------------
; ---- Setting tool (TCP) ----
; TOOL_DATA[1] = {FRAME: X 0.000,Y 0.000,Z 10.000,A 0.000,B 0.000,C 0.000}
$TOOL = {FRAME: X 0.000,Y 0.000,Z 10.000,A 0.000,B 0.000,C 0.000}
; $TOOL = TOOL_DATA[1]
; --------------------------
PTP {A1 -96.25400,A2 -56.15580,A3 114.69800,A4 -12.48820,A5 -62.20070,A6 37.93470}
; ---- Setting reference (Base) ----
$BASE = {FRAME: X 0.000,Y 0.000,Z 0.000,A 0.000,B 0.000,C 0.000}
; --------------------------
; ---- Setting tool (TCP) ----
; TOOL_DATA[1] = {FRAME: X 0.000,Y 0.000,Z 10.000,A 0.000,B 0.000,C 0.000}
$TOOL = {FRAME: X 0.000,Y 0.000,Z 10.000,A 0.000,B 0.000,C 0.000}
; $TOOL = TOOL_DATA[1]
; --------------------------
PTP {A1 -96.25400,A2 -56.15580,A3 114.69800,A4 -12.48820,A5 -62.20070,A6 7.93472}
; ---- Setting reference (Base) ----
$BASE = {FRAME: X 0.000,Y 0.000,Z 0.000,A 0.000,B 0.000,C 0.000}
; --------------------------
; ---- Setting tool (TCP) ----
; TOOL_DATA[1] = {FRAME: X 0.000,Y 0.000,Z 10.000,A 0.000,B 0.000,C 0.000}
$TOOL = {FRAME: X 0.000,Y 0.000,Z 10.000,A 0.000,B 0.000,C 0.000}
; $TOOL = TOOL_DATA[1]
; --------------------------
PTP {A1 -85.40280,A2 -55.58880,A3 116.29500,A4 -0.21382,A5 -63.73790,A6 1.55082}
; ---- Setting reference (Base) ----
$BASE = {FRAME: X 0.000,Y 0.000,Z 0.000,A 0.000,B 0.000,C 0.000}
; --------------------------
; ---- Setting tool (TCP) ----
; TOOL_DATA[1] = {FRAME: X 0.000,Y 0.000,Z 10.000,A 0.000,B 0.000,C 0.000}
$TOOL = {FRAME: X 0.000,Y 0.000,Z 10.000,A 0.000,B 0.000,C 0.000}
; $TOOL = TOOL_DATA[1]
; --------------------------
PTP {A1 -90.37440,A2 -54.36160,A3 113.66900,A4 -38.20870,A5 -68.52430,A6 18.17120}
; ---- Setting reference (Base) ----
$BASE = {FRAME: X 0.000,Y 0.000,Z 0.000,A 0.000,B 0.000,C 0.000}
; --------------------------
; ---- Setting tool (TCP) ----
; TOOL_DATA[1] = {FRAME: X 0.000,Y 0.000,Z 10.000,A 0.000,B 0.000,C 0.000}
$TOOL = {FRAME: X 0.000,Y 0.000,Z 10.000,A 0.000,B 0.000,C 0.000}
; $TOOL = TOOL_DATA[1]
; --------------------------
PTP {A1 -80.41830,A2 -54.74870,A3 113.77000,A4 38.35930,A5 -66.79860,A6 -15.87110}
; ---- Setting reference (Base) ----
$BASE = {FRAME: X 0.000,Y 0.000,Z 0.000,A 0.000,B 0.000,C 0.000}
; --------------------------
; ---- Setting tool (TCP) ----
; TOOL_DATA[1] = {FRAME: X 0.000,Y 0.000,Z 10.000,A 0.000,B 0.000,C 0.000}
$TOOL = {FRAME: X 0.000,Y 0.000,Z 10.000,A 0.000,B 0.000,C 0.000}
; $TOOL = TOOL_DATA[1]
; --------------------------
PTP {A1 -85.40280,A2 -55.58880,A3 116.29500,A4 -0.21382,A5 -63.73790,A6 1.55082}
; ---- Setting reference (Base) ----
$BASE = {FRAME: X 0.000,Y 0.000,Z 0.000,A 0.000,B 0.000,C 0.000}
; --------------------------
; ---- Setting tool (TCP) ----
; TOOL_DATA[1] = {FRAME: X 0.000,Y 0.000,Z 10.000,A 0.000,B 0.000,C 0.000}
$TOOL = {FRAME: X 0.000,Y 0.000,Z 10.000,A 0.000,B 0.000,C 0.000}
; $TOOL = TOOL_DATA[1]
; --------------------------
PTP {A1 -85.40280,A2 -55.58880,A3 116.29500,A4 -0.21382,A5 -63.73790,A6 -28.44920}
; ---- Setting reference (Base) ----
$BASE = {FRAME: X 0.000,Y 0.000,Z 0.000,A 0.000,B 0.000,C 0.000}
; --------------------------
; ---- Setting tool (TCP) ----
; TOOL_DATA[1] = {FRAME: X 0.000,Y 0.000,Z 10.000,A 0.000,B 0.000,C 0.000}
$TOOL = {FRAME: X 0.000,Y 0.000,Z 10.000,A 0.000,B 0.000,C 0.000}
; $TOOL = TOOL_DATA[1]
; --------------------------
PTP {A1 -85.40280,A2 -55.58880,A3 116.29500,A4 -0.21382,A5 -63.73790,A6 31.55080}
; ---- Setting reference (Base) ----
$BASE = {FRAME: X 0.000,Y 0.000,Z 0.000,A 0.000,B 0.000,C 0.000}
; --------------------------
; ---- Setting tool (TCP) ----
; TOOL_DATA[1] = {FRAME: X 0.000,Y 0.000,Z 10.000,A 0.000,B 0.000,C 0.000}
$TOOL = {FRAME: X 0.000,Y 0.000,Z 10.000,A 0.000,B 0.000,C 0.000}
; $TOOL = TOOL_DATA[1]
; --------------------------
PTP {A1 -85.40280,A2 -55.58880,A3 116.29500,A4 -0.21382,A5 -63.73790,A6 1.55082}
; ---- Setting reference (Base) ----
$BASE = {FRAME: X 0.000,Y 0.000,Z 0.000,A 0.000,B 0.000,C 0.000}
; --------------------------
; ---- Setting tool (TCP) ----
; TOOL_DATA[1] = {FRAME: X 0.000,Y 0.000,Z 10.000,A 0.000,B 0.000,C 0.000}
$TOOL = {FRAME: X 0.000,Y 0.000,Z 10.000,A 0.000,B 0.000,C 0.000}
; $TOOL = TOOL_DATA[1]
; --------------------------
PTP {A1 -86.61910,A2 -55.53200,A3 116.26200,A4 -1.56781,A5 -63.77090,A6 2.21360}
; ---- Setting reference (Base) ----
$BASE = {FRAME: X 0.000,Y 0.000,Z 0.000,A 0.000,B 0.000,C 0.000}
; --------------------------
; ---- Setting tool (TCP) ----
; TOOL_DATA[1] = {FRAME: X 0.000,Y 0.000,Z 10.000,A 0.000,B 0.000,C 0.000}
$TOOL = {FRAME: X 0.000,Y 0.000,Z 10.000,A 0.000,B 0.000,C 0.000}
; $TOOL = TOOL_DATA[1]
; --------------------------
PTP {A1 -91.55040,A2 -54.23060,A3 113.46400,A4 -39.42040,A5 -68.84330,A6 18.72360}
; ---- Setting reference (Base) ----
$BASE = {FRAME: X 0.000,Y 0.000,Z 0.000,A 0.000,B 0.000,C 0.000}
; --------------------------
; ---- Setting tool (TCP) ----
; TOOL_DATA[1] = {FRAME: X 0.000,Y 0.000,Z 10.000,A 0.000,B 0.000,C 0.000}
$TOOL = {FRAME: X 0.000,Y 0.000,Z 10.000,A 0.000,B 0.000,C 0.000}
; $TOOL = TOOL_DATA[1]
; --------------------------
PTP {A1 -81.60040,A2 -54.77020,A3 113.91000,A4 37.10660,A5 -66.52090,A6 -15.26880}
; ---- Setting reference (Base) ----
$BASE = {FRAME: X 0.000,Y 0.000,Z 0.000,A 0.000,B 0.000,C 0.000}
; --------------------------
; ---- Setting tool (TCP) ----
; TOOL_DATA[1] = {FRAME: X 0.000,Y 0.000,Z 10.000,A 0.000,B 0.000,C 0.000}
$TOOL = {FRAME: X 0.000,Y 0.000,Z 10.000,A 0.000,B 0.000,C 0.000}
; $TOOL = TOOL_DATA[1]
; --------------------------
PTP {A1 -86.61910,A2 -55.53200,A3 116.26200,A4 -1.56781,A5 -63.77090,A6 2.21360}
; ---- Setting reference (Base) ----
$BASE = {FRAME: X 0.000,Y 0.000,Z 0.000,A 0.000,B 0.000,C 0.000}
; --------------------------
; ---- Setting tool (TCP) ----
; TOOL_DATA[1] = {FRAME: X 0.000,Y 0.000,Z 10.000,A 0.000,B 0.000,C 0.000}
$TOOL = {FRAME: X 0.000,Y 0.000,Z 10.000,A 0.000,B 0.000,C 0.000}
; $TOOL = TOOL_DATA[1]
; --------------------------
PTP {A1 -86.61910,A2 -55.53200,A3 116.26200,A4 -1.56781,A5 -63.77090,A6 -27.78640}
; ---- Setting reference (Base) ----
$BASE = {FRAME: X 0.000,Y 0.000,Z 0.000,A 0.000,B 0.000,C 0.000}
; --------------------------
; ---- Setting tool (TCP) ----
; TOOL_DATA[1] = {FRAME: X 0.000,Y 0.000,Z 10.000,A 0.000,B 0.000,C 0.000}
$TOOL = {FRAME: X 0.000,Y 0.000,Z 10.000,A 0.000,B 0.000,C 0.000}
; $TOOL = TOOL_DATA[1]
; --------------------------
PTP {A1 -86.61910,A2 -55.53200,A3 116.26200,A4 -1.56781,A5 -63.77090,A6 32.21360}
; ---- Setting reference (Base) ----
$BASE = {FRAME: X 0.000,Y 0.000,Z 0.000,A 0.000,B 0.000,C 0.000}
; --------------------------
; ---- Setting tool (TCP) ----
; TOOL_DATA[1] = {FRAME: X 0.000,Y 0.000,Z 10.000,A 0.000,B 0.000,C 0.000}
$TOOL = {FRAME: X 0.000,Y 0.000,Z 10.000,A 0.000,B 0.000,C 0.000}
; $TOOL = TOOL_DATA[1]
; --------------------------
PTP {A1 -86.61910,A2 -55.53200,A3 116.26200,A4 -1.56781,A5 -63.77090,A6 2.21360}
; ---- Setting reference (Base) ----
$BASE = {FRAME: X 0.000,Y 0.000,Z 0.000,A 0.000,B 0.000,C 0.000}
; --------------------------
; ---- Setting tool (TCP) ----
; TOOL_DATA[1] = {FRAME: X 0.000,Y 0.000,Z 10.000,A 0.000,B 0.000,C 0.000}
$TOOL = {FRAME: X 0.000,Y 0.000,Z 10.000,A 0.000,B 0.000,C 0.000}
; $TOOL = TOOL_DATA[1]
; --------------------------
PTP {A1 -87.83410,A2 -55.45720,A3 116.18700,A4 -2.91995,A5 -63.79430,A6 2.87523}
; ---- Setting reference (Base) ----
$BASE = {FRAME: X 0.000,Y 0.000,Z 0.000,A 0.000,B 0.000,C 0.000}
; --------------------------
; ---- Setting tool (TCP) ----
; TOOL_DATA[1] = {FRAME: X 0.000,Y 0.000,Z 10.000,A 0.000,B 0.000,C 0.000}
$TOOL = {FRAME: X 0.000,Y 0.000,Z 10.000,A 0.000,B 0.000,C 0.000}
; $TOOL = TOOL_DATA[1]
; --------------------------
PTP {A1 -92.72090,A2 -54.08170,A3 113.21800,A4 -40.62590,A5 -69.15460,A6 19.28230}
; ---- Setting reference (Base) ----
$BASE = {FRAME: X 0.000,Y 0.000,Z 0.000,A 0.000,B 0.000,C 0.000}
; --------------------------
; ---- Setting tool (TCP) ----
; TOOL_DATA[1] = {FRAME: X 0.000,Y 0.000,Z 10.000,A 0.000,B 0.000,C 0.000}
$TOOL = {FRAME: X 0.000,Y 0.000,Z 10.000,A 0.000,B 0.000,C 0.000}
; $TOOL = TOOL_DATA[1]
; --------------------------
PTP {A1 -82.78550,A2 -54.77340,A3 114.00900,A4 35.85030,A5 -66.23730,A6 -14.67360}
; ---- Setting reference (Base) ----
$BASE = {FRAME: X 0.000,Y 0.000,Z 0.000,A 0.000,B 0.000,C 0.000}
; --------------------------
; ---- Setting tool (TCP) ----
; TOOL_DATA[1] = {FRAME: X 0.000,Y 0.000,Z 10.000,A 0.000,B 0.000,C 0.000}
$TOOL = {FRAME: X 0.000,Y 0.000,Z 10.000,A 0.000,B 0.000,C 0.000}
; $TOOL = TOOL_DATA[1]
; --------------------------
PTP {A1 -87.83410,A2 -55.45720,A3 116.18700,A4 -2.91995,A5 -63.79430,A6 2.87523}
; ---- Setting reference (Base) ----
$BASE = {FRAME: X 0.000,Y 0.000,Z 0.000,A 0.000,B 0.000,C 0.000}
; --------------------------
; ---- Setting tool (TCP) ----
; TOOL_DATA[1] = {FRAME: X 0.000,Y 0.000,Z 10.000,A 0.000,B 0.000,C 0.000}
$TOOL = {FRAME: X 0.000,Y 0.000,Z 10.000,A 0.000,B 0.000,C 0.000}
; $TOOL = TOOL_DATA[1]
; --------------------------
PTP {A1 -87.83410,A2 -55.45720,A3 116.18700,A4 -2.91995,A5 -63.79430,A6 -27.12480}
; ---- Setting reference (Base) ----
$BASE = {FRAME: X 0.000,Y 0.000,Z 0.000,A 0.000,B 0.000,C 0.000}
; --------------------------
; ---- Setting tool (TCP) ----
; TOOL_DATA[1] = {FRAME: X 0.000,Y 0.000,Z 10.000,A 0.000,B 0.000,C 0.000}
$TOOL = {FRAME: X 0.000,Y 0.000,Z 10.000,A 0.000,B 0.000,C 0.000}
; $TOOL = TOOL_DATA[1]
; --------------------------
PTP {A1 -87.83410,A2 -55.45720,A3 116.18700,A4 -2.91995,A5 -63.79430,A6 32.87520}
; ---- Setting reference (Base) ----
$BASE = {FRAME: X 0.000,Y 0.000,Z 0.000,A 0.000,B 0.000,C 0.000}
; --------------------------
; ---- Setting tool (TCP) ----
; TOOL_DATA[1] = {FRAME: X 0.000,Y 0.000,Z 10.000,A 0.000,B 0.000,C 0.000}
$TOOL = {FRAME: X 0.000,Y 0.000,Z 10.000,A 0.000,B 0.000,C 0.000}
; $TOOL = TOOL_DATA[1]
; --------------------------
PTP {A1 -87.83410,A2 -55.45720,A3 116.18700,A4 -2.91995,A5 -63.79430,A6 2.87523}
; ---- Setting reference (Base) ----
$BASE = {FRAME: X 0.000,Y 0.000,Z 0.000,A 0.000,B 0.000,C 0.000}
; --------------------------
; ---- Setting tool (TCP) ----
; TOOL_DATA[1] = {FRAME: X 0.000,Y 0.000,Z 10.000,A 0.000,B 0.000,C 0.000}
$TOOL = {FRAME: X 0.000,Y 0.000,Z 10.000,A 0.000,B 0.000,C 0.000}
; $TOOL = TOOL_DATA[1]
; --------------------------
PTP {A1 -89.04660,A2 -55.36440,A3 116.07100,A4 -4.26952,A5 -63.80810,A6 3.53652}
; ---- Setting reference (Base) ----
$BASE = {FRAME: X 0.000,Y 0.000,Z 0.000,A 0.000,B 0.000,C 0.000}
; --------------------------
; ---- Setting tool (TCP) ----
; TOOL_DATA[1] = {FRAME: X 0.000,Y 0.000,Z 10.000,A 0.000,B 0.000,C 0.000}
$TOOL = {FRAME: X 0.000,Y 0.000,Z 10.000,A 0.000,B 0.000,C 0.000}
; $TOOL = TOOL_DATA[1]
; --------------------------
PTP {A1 -93.88520,A2 -53.91510,A3 112.93200,A4 -41.82450,A5 -69.45860,A6 19.84780}
; ---- Setting reference (Base) ----
$BASE = {FRAME: X 0.000,Y 0.000,Z 0.000,A 0.000,B 0.000,C 0.000}
; --------------------------
; ---- Setting tool (TCP) ----
; TOOL_DATA[1] = {FRAME: X 0.000,Y 0.000,Z 10.000,A 0.000,B 0.000,C 0.000}
$TOOL = {FRAME: X 0.000,Y 0.000,Z 10.000,A 0.000,B 0.000,C 0.000}
; $TOOL = TOOL_DATA[1]
; --------------------------
PTP {A1 -83.97260,A2 -54.75810,A3 114.06700,A4 34.59140,A5 -65.94740,A6 -14.08540}
; ---- Setting reference (Base) ----
$BASE = {FRAME: X 0.000,Y 0.000,Z 0.000,A 0.000,B 0.000,C 0.000}
; --------------------------
; ---- Setting tool (TCP) ----
; TOOL_DATA[1] = {FRAME: X 0.000,Y 0.000,Z 10.000,A 0.000,B 0.000,C 0.000}
$TOOL = {FRAME: X 0.000,Y 0.000,Z 10.000,A 0.000,B 0.000,C 0.000}
; $TOOL = TOOL_DATA[1]
; --------------------------
PTP {A1 -89.04660,A2 -55.36440,A3 116.07100,A4 -4.26952,A5 -63.80810,A6 3.53652}
; ---- Setting reference (Base) ----
$BASE = {FRAME: X 0.000,Y 0.000,Z 0.000,A 0.000,B 0.000,C 0.000}
; --------------------------
; ---- Setting tool (TCP) ----
; TOOL_DATA[1] = {FRAME: X 0.000,Y 0.000,Z 10.000,A 0.000,B 0.000,C 0.000}
$TOOL = {FRAME: X 0.000,Y 0.000,Z 10.000,A 0.000,B 0.000,C 0.000}
; $TOOL = TOOL_DATA[1]
; --------------------------
PTP {A1 -89.04660,A2 -55.36440,A3 116.07100,A4 -4.26952,A5 -63.80810,A6 -26.46350}
; ---- Setting reference (Base) ----
$BASE = {FRAME: X 0.000,Y 0.000,Z 0.000,A 0.000,B 0.000,C 0.000}
; --------------------------
; ---- Setting tool (TCP) ----
; TOOL_DATA[1] = {FRAME: X 0.000,Y 0.000,Z 10.000,A 0.000,B 0.000,C 0.000}
$TOOL = {FRAME: X 0.000,Y 0.000,Z 10.000,A 0.000,B 0.000,C 0.000}
; $TOOL = TOOL_DATA[1]
; --------------------------
PTP {A1 -89.04660,A2 -55.36440,A3 116.07100,A4 -4.26952,A5 -63.80810,A6 33.53650}
; ---- Setting reference (Base) ----
$BASE = {FRAME: X 0.000,Y 0.000,Z 0.000,A 0.000,B 0.000,C 0.000}
; --------------------------
; ---- Setting tool (TCP) ----
; TOOL_DATA[1] = {FRAME: X 0.000,Y 0.000,Z 10.000,A 0.000,B 0.000,C 0.000}
$TOOL = {FRAME: X 0.000,Y 0.000,Z 10.000,A 0.000,B 0.000,C 0.000}
; $TOOL = TOOL_DATA[1]
; --------------------------
PTP {A1 -89.04660,A2 -55.36440,A3 116.07100,A4 -4.26952,A5 -63.80810,A6 3.53652}
; ---- Setting reference (Base) ----
$BASE = {FRAME: X 0.000,Y 0.000,Z 0.000,A 0.000,B 0.000,C 0.000}
; --------------------------
; ---- Setting tool (TCP) ----
; TOOL_DATA[1] = {FRAME: X 0.000,Y 0.000,Z 10.000,A 0.000,B 0.000,C 0.000}
$TOOL = {FRAME: X 0.000,Y 0.000,Z 10.000,A 0.000,B 0.000,C 0.000}
; $TOOL = TOOL_DATA[1]
; --------------------------
PTP {A1 -90.25570,A2 -55.25360,A3 115.91300,A4 -5.61579,A5 -63.81230,A6 4.19830}
; ---- Setting reference (Base) ----
$BASE = {FRAME: X 0.000,Y 0.000,Z 0.000,A 0.000,B 0.000,C 0.000}
; --------------------------
; ---- Setting tool (TCP) ----
; TOOL_DATA[1] = {FRAME: X 0.000,Y 0.000,Z 10.000,A 0.000,B 0.000,C 0.000}
$TOOL = {FRAME: X 0.000,Y 0.000,Z 10.000,A 0.000,B 0.000,C 0.000}
; $TOOL = TOOL_DATA[1]
; --------------------------
PTP {A1 -95.04220,A2 -53.73080,A3 112.60500,A4 -43.01530,A5 -69.75580,A6 20.42070}
; ---- Setting reference (Base) ----
$BASE = {FRAME: X 0.000,Y 0.000,Z 0.000,A 0.000,B 0.000,C 0.000}
; --------------------------
; ---- Setting tool (TCP) ----
; TOOL_DATA[1] = {FRAME: X 0.000,Y 0.000,Z 10.000,A 0.000,B 0.000,C 0.000}
$TOOL = {FRAME: X 0.000,Y 0.000,Z 10.000,A 0.000,B 0.000,C 0.000}
; $TOOL = TOOL_DATA[1]
; --------------------------
PTP {A1 -85.16070,A2 -54.72460,A3 114.08400,A4 33.33090,A5 -65.65070,A6 -13.50350}
; ---- Setting reference (Base) ----
$BASE = {FRAME: X 0.000,Y 0.000,Z 0.000,A 0.000,B 0.000,C 0.000}
; --------------------------
; ---- Setting tool (TCP) ----
; TOOL_DATA[1] = {FRAME: X 0.000,Y 0.000,Z 10.000,A 0.000,B 0.000,C 0.000}
$TOOL = {FRAME: X 0.000,Y 0.000,Z 10.000,A 0.000,B 0.000,C 0.000}
; $TOOL = TOOL_DATA[1]
; --------------------------
PTP {A1 -90.25570,A2 -55.25360,A3 115.91300,A4 -5.61579,A5 -63.81230,A6 4.19830}
; ---- Setting reference (Base) ----
$BASE = {FRAME: X 0.000,Y 0.000,Z 0.000,A 0.000,B 0.000,C 0.000}
; --------------------------
; ---- Setting tool (TCP) ----
; TOOL_DATA[1] = {FRAME: X 0.000,Y 0.000,Z 10.000,A 0.000,B 0.000,C 0.000}
$TOOL = {FRAME: X 0.000,Y 0.000,Z 10.000,A 0.000,B 0.000,C 0.000}
; $TOOL = TOOL_DATA[1]
; --------------------------
PTP {A1 -90.25570,A2 -55.25360,A3 115.91300,A4 -5.61579,A5 -63.81230,A6 -25.80170}
; ---- Setting reference (Base) ----
$BASE = {FRAME: X 0.000,Y 0.000,Z 0.000,A 0.000,B 0.000,C 0.000}
; --------------------------
; ---- Setting tool (TCP) ----
; TOOL_DATA[1] = {FRAME: X 0.000,Y 0.000,Z 10.000,A 0.000,B 0.000,C 0.000}
$TOOL = {FRAME: X 0.000,Y 0.000,Z 10.000,A 0.000,B 0.000,C 0.000}
; $TOOL = TOOL_DATA[1]
; --------------------------
PTP {A1 -90.25570,A2 -55.25360,A3 115.91300,A4 -5.61579,A5 -63.81230,A6 34.19830}
; ---- Setting reference (Base) ----
$BASE = {FRAME: X 0.000,Y 0.000,Z 0.000,A 0.000,B 0.000,C 0.000}
; --------------------------
; ---- Setting tool (TCP) ----
; TOOL_DATA[1] = {FRAME: X 0.000,Y 0.000,Z 10.000,A 0.000,B 0.000,C 0.000}
$TOOL = {FRAME: X 0.000,Y 0.000,Z 10.000,A 0.000,B 0.000,C 0.000}
; $TOOL = TOOL_DATA[1]
; --------------------------
PTP {A1 -90.25570,A2 -55.25360,A3 115.91300,A4 -5.61579,A5 -63.81230,A6 4.19830}
; ---- Setting reference (Base) ----
$BASE = {FRAME: X 0.000,Y 0.000,Z 0.000,A 0.000,B 0.000,C 0.000}
; --------------------------
; ---- Setting tool (TCP) ----
; TOOL_DATA[1] = {FRAME: X 0.000,Y 0.000,Z 10.000,A 0.000,B 0.000,C 0.000}
$TOOL = {FRAME: X 0.000,Y 0.000,Z 10.000,A 0.000,B 0.000,C 0.000}
; $TOOL = TOOL_DATA[1]
; --------------------------
PTP {A1 -91.46010,A2 -55.12500,A3 115.71400,A4 -6.95807,A5 -63.80680,A6 4.86139}
; ---- Setting reference (Base) ----
$BASE = {FRAME: X 0.000,Y 0.000,Z 0.000,A 0.000,B 0.000,C 0.000}
; --------------------------
; ---- Setting tool (TCP) ----
; TOOL_DATA[1] = {FRAME: X 0.000,Y 0.000,Z 10.000,A 0.000,B 0.000,C 0.000}
$TOOL = {FRAME: X 0.000,Y 0.000,Z 10.000,A 0.000,B 0.000,C 0.000}
; $TOOL = TOOL_DATA[1]
; --------------------------
PTP {A1 -96.19110,A2 -53.52900,A3 112.23700,A4 -44.19750,A5 -70.04650,A6 21.00130}
; ---- Setting reference (Base) ----
$BASE = {FRAME: X 0.000,Y 0.000,Z 0.000,A 0.000,B 0.000,C 0.000}
; --------------------------
; ---- Setting tool (TCP) ----
; TOOL_DATA[1] = {FRAME: X 0.000,Y 0.000,Z 10.000,A 0.000,B 0.000,C 0.000}
$TOOL = {FRAME: X 0.000,Y 0.000,Z 10.000,A 0.000,B 0.000,C 0.000}
; $TOOL = TOOL_DATA[1]
; --------------------------
PTP {A1 -86.34880,A2 -54.67280,A3 114.06000,A4 32.06970,A5 -65.34680,A6 -12.92740}
; ---- Setting reference (Base) ----
$BASE = {FRAME: X 0.000,Y 0.000,Z 0.000,A 0.000,B 0.000,C 0.000}
; --------------------------
; ---- Setting tool (TCP) ----
; TOOL_DATA[1] = {FRAME: X 0.000,Y 0.000,Z 10.000,A 0.000,B 0.000,C 0.000}
$TOOL = {FRAME: X 0.000,Y 0.000,Z 10.000,A 0.000,B 0.000,C 0.000}
; $TOOL = TOOL_DATA[1]
; --------------------------
PTP {A1 -91.46010,A2 -55.12500,A3 115.71400,A4 -6.95807,A5 -63.80680,A6 4.86139}
; ---- Setting reference (Base) ----
$BASE = {FRAME: X 0.000,Y 0.000,Z 0.000,A 0.000,B 0.000,C 0.000}
; --------------------------
; ---- Setting tool (TCP) ----
; TOOL_DATA[1] = {FRAME: X 0.000,Y 0.000,Z 10.000,A 0.000,B 0.000,C 0.000}
$TOOL = {FRAME: X 0.000,Y 0.000,Z 10.000,A 0.000,B 0.000,C 0.000}
; $TOOL = TOOL_DATA[1]
; --------------------------
PTP {A1 -91.46010,A2 -55.12500,A3 115.71400,A4 -6.95807,A5 -63.80680,A6 -25.13860}
; ---- Setting reference (Base) ----
$BASE = {FRAME: X 0.000,Y 0.000,Z 0.000,A 0.000,B 0.000,C 0.000}
; --------------------------
; ---- Setting tool (TCP) ----
; TOOL_DATA[1] = {FRAME: X 0.000,Y 0.000,Z 10.000,A 0.000,B 0.000,C 0.000}
$TOOL = {FRAME: X 0.000,Y 0.000,Z 10.000,A 0.000,B 0.000,C 0.000}
; $TOOL = TOOL_DATA[1]
; --------------------------
PTP {A1 -91.46010,A2 -55.12500,A3 115.71400,A4 -6.95807,A5 -63.80680,A6 34.86140}
; ---- Setting reference (Base) ----
$BASE = {FRAME: X 0.000,Y 0.000,Z 0.000,A 0.000,B 0.000,C 0.000}
; --------------------------
; ---- Setting tool (TCP) ----
; TOOL_DATA[1] = {FRAME: X 0.000,Y 0.000,Z 10.000,A 0.000,B 0.000,C 0.000}
$TOOL = {FRAME: X 0.000,Y 0.000,Z 10.000,A 0.000,B 0.000,C 0.000}
; $TOOL = TOOL_DATA[1]
; --------------------------
PTP {A1 -91.46010,A2 -55.12500,A3 115.71400,A4 -6.95807,A5 -63.80680,A6 4.86139}
; ---- Setting reference (Base) ----
$BASE = {FRAME: X 0.000,Y 0.000,Z 0.000,A 0.000,B 0.000,C 0.000}
; --------------------------
; ---- Setting tool (TCP) ----
; TOOL_DATA[1] = {FRAME: X 0.000,Y 0.000,Z 10.000,A 0.000,B 0.000,C 0.000}
$TOOL = {FRAME: X 0.000,Y 0.000,Z 10.000,A 0.000,B 0.000,C 0.000}
; $TOOL = TOOL_DATA[1]
; --------------------------
PTP {A1 -92.65900,A2 -54.97860,A3 115.47300,A4 -8.29569,A5 -63.79180,A6 5.52662}
; ---- Setting reference (Base) ----
$BASE = {FRAME: X 0.000,Y 0.000,Z 0.000,A 0.000,B 0.000,C 0.000}
; --------------------------
; ---- Setting tool (TCP) ----
; TOOL_DATA[1] = {FRAME: X 0.000,Y 0.000,Z 10.000,A 0.000,B 0.000,C 0.000}
$TOOL = {FRAME: X 0.000,Y 0.000,Z 10.000,A 0.000,B 0.000,C 0.000}
; $TOOL = TOOL_DATA[1]
; --------------------------
PTP {A1 -97.33100,A2 -53.30950,A3 111.83000,A4 -45.37020,A5 -70.33110,A6 21.59010}
; ---- Setting reference (Base) ----
$BASE = {FRAME: X 0.000,Y 0.000,Z 0.000,A 0.000,B 0.000,C 0.000}
; --------------------------
; ---- Setting tool (TCP) ----
; TOOL_DATA[1] = {FRAME: X 0.000,Y 0.000,Z 10.000,A 0.000,B 0.000,C 0.000}
$TOOL = {FRAME: X 0.000,Y 0.000,Z 10.000,A 0.000,B 0.000,C 0.000}
; $TOOL = TOOL_DATA[1]
; --------------------------
PTP {A1 -87.53580,A2 -54.60290,A3 113.99400,A4 30.80860,A5 -65.03530,A6 -12.35680}
; ---- Setting reference (Base) ----
$BASE = {FRAME: X 0.000,Y 0.000,Z 0.000,A 0.000,B 0.000,C 0.000}
; --------------------------
; ---- Setting tool (TCP) ----
; TOOL_DATA[1] = {FRAME: X 0.000,Y 0.000,Z 10.000,A 0.000,B 0.000,C 0.000}
$TOOL = {FRAME: X 0.000,Y 0.000,Z 10.000,A 0.000,B 0.000,C 0.000}
; $TOOL = TOOL_DATA[1]
; --------------------------
PTP {A1 -92.65900,A2 -54.97860,A3 115.47300,A4 -8.29569,A5 -63.79180,A6 5.52662}
; ---- Setting reference (Base) ----
$BASE = {FRAME: X 0.000,Y 0.000,Z 0.000,A 0.000,B 0.000,C 0.000}
; --------------------------
; ---- Setting tool (TCP) ----
; TOOL_DATA[1] = {FRAME: X 0.000,Y 0.000,Z 10.000,A 0.000,B 0.000,C 0.000}
$TOOL = {FRAME: X 0.000,Y 0.000,Z 10.000,A 0.000,B 0.000,C 0.000}
; $TOOL = TOOL_DATA[1]
; --------------------------
PTP {A1 -92.65900,A2 -54.97860,A3 115.47300,A4 -8.29569,A5 -63.79180,A6 -24.47340}
; ---- Setting reference (Base) ----
$BASE = {FRAME: X 0.000,Y 0.000,Z 0.000,A 0.000,B 0.000,C 0.000}
; --------------------------
; ---- Setting tool (TCP) ----
; TOOL_DATA[1] = {FRAME: X 0.000,Y 0.000,Z 10.000,A 0.000,B 0.000,C 0.000}
$TOOL = {FRAME: X 0.000,Y 0.000,Z 10.000,A 0.000,B 0.000,C 0.000}
; $TOOL = TOOL_DATA[1]
; --------------------------
PTP {A1 -92.65900,A2 -54.97860,A3 115.47300,A4 -8.29569,A5 -63.79180,A6 35.52660}
; ---- Setting reference (Base) ----
$BASE = {FRAME: X 0.000,Y 0.000,Z 0.000,A 0.000,B 0.000,C 0.000}
; --------------------------
; ---- Setting tool (TCP) ----
; TOOL_DATA[1] = {FRAME: X 0.000,Y 0.000,Z 10.000,A 0.000,B 0.000,C 0.000}
$TOOL = {FRAME: X 0.000,Y 0.000,Z 10.000,A 0.000,B 0.000,C 0.000}
; $TOOL = TOOL_DATA[1]
; --------------------------
PTP {A1 -92.65900,A2 -54.97860,A3 115.47300,A4 -8.29569,A5 -63.79180,A6 5.52662}
; ---- Setting reference (Base) ----
$BASE = {FRAME: X 0.000,Y 0.000,Z 0.000,A 0.000,B 0.000,C 0.000}
; --------------------------
; ---- Setting tool (TCP) ----
; TOOL_DATA[1] = {FRAME: X 0.000,Y 0.000,Z 10.000,A 0.000,B 0.000,C 0.000}
$TOOL = {FRAME: X 0.000,Y 0.000,Z 10.000,A 0.000,B 0.000,C 0.000}
; $TOOL = TOOL_DATA[1]
; --------------------------
PTP {A1 -93.85130,A2 -54.81450,A3 115.19200,A4 -9.62798,A5 -63.76730,A6 6.19478}
; ---- Setting reference (Base) ----
$BASE = {FRAME: X 0.000,Y 0.000,Z 0.000,A 0.000,B 0.000,C 0.000}
; --------------------------
; ---- Setting tool (TCP) ----
; TOOL_DATA[1] = {FRAME: X 0.000,Y 0.000,Z 10.000,A 0.000,B 0.000,C 0.000}
$TOOL = {FRAME: X 0.000,Y 0.000,Z 10.000,A 0.000,B 0.000,C 0.000}
; $TOOL = TOOL_DATA[1]
; --------------------------
PTP {A1 -98.46130,A2 -53.07260,A3 111.38200,A4 -46.53270,A5 -70.61010,A6 22.18740}
; ---- Setting reference (Base) ----
$BASE = {FRAME: X 0.000,Y 0.000,Z 0.000,A 0.000,B 0.000,C 0.000}
; --------------------------
; ---- Setting tool (TCP) ----
; TOOL_DATA[1] = {FRAME: X 0.000,Y 0.000,Z 10.000,A 0.000,B 0.000,C 0.000}
$TOOL = {FRAME: X 0.000,Y 0.000,Z 10.000,A 0.000,B 0.000,C 0.000}
; $TOOL = TOOL_DATA[1]
; --------------------------
PTP {A1 -88.72080,A2 -54.51500,A3 113.88800,A4 29.54860,A5 -64.71580,A6 -11.79090}
; ---- Setting reference (Base) ----
$BASE = {FRAME: X 0.000,Y 0.000,Z 0.000,A 0.000,B 0.000,C 0.000}
; --------------------------
; ---- Setting tool (TCP) ----
; TOOL_DATA[1] = {FRAME: X 0.000,Y 0.000,Z 10.000,A 0.000,B 0.000,C 0.000}
$TOOL = {FRAME: X 0.000,Y 0.000,Z 10.000,A 0.000,B 0.000,C 0.000}
; $TOOL = TOOL_DATA[1]
; --------------------------
PTP {A1 -93.85130,A2 -54.81450,A3 115.19200,A4 -9.62798,A5 -63.76730,A6 6.19478}
; ---- Setting reference (Base) ----
$BASE = {FRAME: X 0.000,Y 0.000,Z 0.000,A 0.000,B 0.000,C 0.000}
; --------------------------
; ---- Setting tool (TCP) ----
; TOOL_DATA[1] = {FRAME: X 0.000,Y 0.000,Z 10.000,A 0.000,B 0.000,C 0.000}
$TOOL = {FRAME: X 0.000,Y 0.000,Z 10.000,A 0.000,B 0.000,C 0.000}
; $TOOL = TOOL_DATA[1]
; --------------------------
PTP {A1 -93.85130,A2 -54.81450,A3 115.19200,A4 -9.62798,A5 -63.76730,A6 -23.80520}
; ---- Setting reference (Base) ----
$BASE = {FRAME: X 0.000,Y 0.000,Z 0.000,A 0.000,B 0.000,C 0.000}
; --------------------------
; ---- Setting tool (TCP) ----
; TOOL_DATA[1] = {FRAME: X 0.000,Y 0.000,Z 10.000,A 0.000,B 0.000,C 0.000}
$TOOL = {FRAME: X 0.000,Y 0.000,Z 10.000,A 0.000,B 0.000,C 0.000}
; $TOOL = TOOL_DATA[1]
; --------------------------
PTP {A1 -93.85130,A2 -54.81450,A3 115.19200,A4 -9.62798,A5 -63.76730,A6 36.19480}
; ---- Setting reference (Base) ----
$BASE = {FRAME: X 0.000,Y 0.000,Z 0.000,A 0.000,B 0.000,C 0.000}
; --------------------------
; ---- Setting tool (TCP) ----
; TOOL_DATA[1] = {FRAME: X 0.000,Y 0.000,Z 10.000,A 0.000,B 0.000,C 0.000}
$TOOL = {FRAME: X 0.000,Y 0.000,Z 10.000,A 0.000,B 0.000,C 0.000}
; $TOOL = TOOL_DATA[1]
; --------------------------
PTP {A1 -93.85130,A2 -54.81450,A3 115.19200,A4 -9.62798,A5 -63.76730,A6 6.19478}
; ---- Setting reference (Base) ----
$BASE = {FRAME: X 0.000,Y 0.000,Z 0.000,A 0.000,B 0.000,C 0.000}
; --------------------------
; ---- Setting tool (TCP) ----
; TOOL_DATA[1] = {FRAME: X 0.000,Y 0.000,Z 10.000,A 0.000,B 0.000,C 0.000}
$TOOL = {FRAME: X 0.000,Y 0.000,Z 10.000,A 0.000,B 0.000,C 0.000}
; $TOOL = TOOL_DATA[1]
; --------------------------
PTP {A1 -95.03610,A2 -54.63280,A3 114.86900,A4 -10.95430,A5 -63.73350,A6 6.86666}
; ---- Setting reference (Base) ----
$BASE = {FRAME: X 0.000,Y 0.000,Z 0.000,A 0.000,B 0.000,C 0.000}
; --------------------------
; ---- Setting tool (TCP) ----
; TOOL_DATA[1] = {FRAME: X 0.000,Y 0.000,Z 10.000,A 0.000,B 0.000,C 0.000}
$TOOL = {FRAME: X 0.000,Y 0.000,Z 10.000,A 0.000,B 0.000,C 0.000}
; $TOOL = TOOL_DATA[1]
; --------------------------
PTP {A1 -99.58100,A2 -52.81830,A3 110.89500,A4 -47.68420,A5 -70.88400,A6 22.79370}
; ---- Setting reference (Base) ----
$BASE = {FRAME: X 0.000,Y 0.000,Z 0.000,A 0.000,B 0.000,C 0.000}
; --------------------------
; ---- Setting tool (TCP) ----
; TOOL_DATA[1] = {FRAME: X 0.000,Y 0.000,Z 10.000,A 0.000,B 0.000,C 0.000}
$TOOL = {FRAME: X 0.000,Y 0.000,Z 10.000,A 0.000,B 0.000,C 0.000}
; $TOOL = TOOL_DATA[1]
; --------------------------
PTP {A1 -89.90270,A2 -54.40900,A3 113.74000,A4 28.29040,A5 -64.38780,A6 -11.22930}
; ---- Setting reference (Base) ----
$BASE = {FRAME: X 0.000,Y 0.000,Z 0.000,A 0.000,B 0.000,C 0.000}
; --------------------------
; ---- Setting tool (TCP) ----
; TOOL_DATA[1] = {FRAME: X 0.000,Y 0.000,Z 10.000,A 0.000,B 0.000,C 0.000}
$TOOL = {FRAME: X 0.000,Y 0.000,Z 10.000,A 0.000,B 0.000,C 0.000}
; $TOOL = TOOL_DATA[1]
; --------------------------
PTP {A1 -95.03610,A2 -54.63280,A3 114.86900,A4 -10.95430,A5 -63.73350,A6 6.86666}
; ---- Setting reference (Base) ----
$BASE = {FRAME: X 0.000,Y 0.000,Z 0.000,A 0.000,B 0.000,C 0.000}
; --------------------------
; ---- Setting tool (TCP) ----
; TOOL_DATA[1] = {FRAME: X 0.000,Y 0.000,Z 10.000,A 0.000,B 0.000,C 0.000}
$TOOL = {FRAME: X 0.000,Y 0.000,Z 10.000,A 0.000,B 0.000,C 0.000}
; $TOOL = TOOL_DATA[1]
; --------------------------
PTP {A1 -95.03610,A2 -54.63280,A3 114.86900,A4 -10.95430,A5 -63.73350,A6 -23.13330}
; ---- Setting reference (Base) ----
$BASE = {FRAME: X 0.000,Y 0.000,Z 0.000,A 0.000,B 0.000,C 0.000}
; --------------------------
; ---- Setting tool (TCP) ----
; TOOL_DATA[1] = {FRAME: X 0.000,Y 0.000,Z 10.000,A 0.000,B 0.000,C 0.000}
$TOOL = {FRAME: X 0.000,Y 0.000,Z 10.000,A 0.000,B 0.000,C 0.000}
; $TOOL = TOOL_DATA[1]
; --------------------------
PTP {A1 -95.03610,A2 -54.63280,A3 114.86900,A4 -10.95430,A5 -63.73350,A6 36.86670}
; ---- Setting reference (Base) ----
$BASE = {FRAME: X 0.000,Y 0.000,Z 0.000,A 0.000,B 0.000,C 0.000}
; --------------------------
; ---- Setting tool (TCP) ----
; TOOL_DATA[1] = {FRAME: X 0.000,Y 0.000,Z 10.000,A 0.000,B 0.000,C 0.000}
$TOOL = {FRAME: X 0.000,Y 0.000,Z 10.000,A 0.000,B 0.000,C 0.000}
; $TOOL = TOOL_DATA[1]
; --------------------------
PTP {A1 -95.03610,A2 -54.63280,A3 114.86900,A4 -10.95430,A5 -63.73350,A6 6.86666}
; ---- Setting reference (Base) ----
$BASE = {FRAME: X 0.000,Y 0.000,Z 0.000,A 0.000,B 0.000,C 0.000}
; --------------------------
; ---- Setting tool (TCP) ----
; TOOL_DATA[1] = {FRAME: X 0.000,Y 0.000,Z 10.000,A 0.000,B 0.000,C 0.000}
$TOOL = {FRAME: X 0.000,Y 0.000,Z 10.000,A 0.000,B 0.000,C 0.000}
; $TOOL = TOOL_DATA[1]
; --------------------------
PTP {A1 -96.21230,A2 -54.43350,A3 114.50600,A4 -12.27410,A5 -63.69060,A6 7.54304}
; ---- Setting reference (Base) ----
$BASE = {FRAME: X 0.000,Y 0.000,Z 0.000,A 0.000,B 0.000,C 0.000}
; --------------------------
; ---- Setting tool (TCP) ----
; TOOL_DATA[1] = {FRAME: X 0.000,Y 0.000,Z 10.000,A 0.000,B 0.000,C 0.000}
$TOOL = {FRAME: X 0.000,Y 0.000,Z 10.000,A 0.000,B 0.000,C 0.000}
; $TOOL = TOOL_DATA[1]
; --------------------------
PTP {A1 -100.69000,A2 -52.54660,A3 110.36800,A4 -48.82410,A5 -71.15310,A6 23.40910}
; ---- Setting reference (Base) ----
$BASE = {FRAME: X 0.000,Y 0.000,Z 0.000,A 0.000,B 0.000,C 0.000}
; --------------------------
; ---- Setting tool (TCP) ----
; TOOL_DATA[1] = {FRAME: X 0.000,Y 0.000,Z 10.000,A 0.000,B 0.000,C 0.000}
$TOOL = {FRAME: X 0.000,Y 0.000,Z 10.000,A 0.000,B 0.000,C 0.000}
; $TOOL = TOOL_DATA[1]
; --------------------------
PTP {A1 -91.08060,A2 -54.28510,A3 113.55100,A4 27.03490,A5 -64.05120,A6 -10.67120}
; ---- Setting reference (Base) ----
$BASE = {FRAME: X 0.000,Y 0.000,Z 0.000,A 0.000,B 0.000,C 0.000}
; --------------------------
; ---- Setting tool (TCP) ----
; TOOL_DATA[1] = {FRAME: X 0.000,Y 0.000,Z 10.000,A 0.000,B 0.000,C 0.000}
$TOOL = {FRAME: X 0.000,Y 0.000,Z 10.000,A 0.000,B 0.000,C 0.000}
; $TOOL = TOOL_DATA[1]
; --------------------------
PTP {A1 -96.21230,A2 -54.43350,A3 114.50600,A4 -12.27410,A5 -63.69060,A6 7.54304}
; ---- Setting reference (Base) ----
$BASE = {FRAME: X 0.000,Y 0.000,Z 0.000,A 0.000,B 0.000,C 0.000}
; --------------------------
; ---- Setting tool (TCP) ----
; TOOL_DATA[1] = {FRAME: X 0.000,Y 0.000,Z 10.000,A 0.000,B 0.000,C 0.000}
$TOOL = {FRAME: X 0.000,Y 0.000,Z 10.000,A 0.000,B 0.000,C 0.000}
; $TOOL = TOOL_DATA[1]
; --------------------------
PTP {A1 -96.21230,A2 -54.43350,A3 114.50600,A4 -12.27410,A5 -63.69060,A6 -22.45700}
; ---- Setting reference (Base) ----
$BASE = {FRAME: X 0.000,Y 0.000,Z 0.000,A 0.000,B 0.000,C 0.000}
; --------------------------
; ---- Setting tool (TCP) ----
; TOOL_DATA[1] = {FRAME: X 0.000,Y 0.000,Z 10.000,A 0.000,B 0.000,C 0.000}
$TOOL = {FRAME: X 0.000,Y 0.000,Z 10.000,A 0.000,B 0.000,C 0.000}
; $TOOL = TOOL_DATA[1]
; --------------------------
PTP {A1 -96.21230,A2 -54.43350,A3 114.50600,A4 -12.27410,A5 -63.69060,A6 37.54300}
; ---- Setting reference (Base) ----
$BASE = {FRAME: X 0.000,Y 0.000,Z 0.000,A 0.000,B 0.000,C 0.000}
; --------------------------
; ---- Setting tool (TCP) ----
; TOOL_DATA[1] = {FRAME: X 0.000,Y 0.000,Z 10.000,A 0.000,B 0.000,C 0.000}
$TOOL = {FRAME: X 0.000,Y 0.000,Z 10.000,A 0.000,B 0.000,C 0.000}
; $TOOL = TOOL_DATA[1]
; --------------------------
PTP {A1 -96.21230,A2 -54.43350,A3 114.50600,A4 -12.27410,A5 -63.69060,A6 7.54304}
; ---- Setting reference (Base) ----
$BASE = {FRAME: X 0.000,Y 0.000,Z 0.000,A 0.000,B 0.000,C 0.000}
; --------------------------
; ---- Setting tool (TCP) ----
; TOOL_DATA[1] = {FRAME: X 0.000,Y 0.000,Z 10.000,A 0.000,B 0.000,C 0.000}
$TOOL = {FRAME: X 0.000,Y 0.000,Z 10.000,A 0.000,B 0.000,C 0.000}
; $TOOL = TOOL_DATA[1]
; --------------------------
PTP {A1 -91.61000,A2 -62.00000,A3 116.14000,A4 -7.59000,A5 -57.42000,A6 5.89000}
END
